FUNCTION_BLOCK FB_DelaySampling
VAR_INPUT
	udiDelaySampling	: UDINT;
	diData				: DINT;
END_VAR
VAR_OUTPUT
	diOutData		: DINT;
END_VAR
VAR
	i				: UDINT;
	diDelayData		: ARRAY[0..1000] OF DINT;
END_VAR

//Get latest data
diDelayData[0]:=diData;

//Slide window
FOR i:=udiDelaySampling TO 1 BY -1 DO
	diDelayData[i] := diDelayData[i -1];
END_FOR

diOutData := diDelayData[udiDelaySampling];

END_FUNCTION_BLOCK

(* stored: Version 1.1.0.1
   POU FB_DelaySampling: Id {ef17dc93-d612-4d7e-93b1-556a8a6188ca}, SpecialFunc None *)
